Staubli VAL3: xyPut.pgx

program xyPut(num x_nX (dimensions=1), num x_nY (dimensions=1), string x_sKey (dimensions=1))
begin
  gotoxy(x_nX,x_nY)
  put(x_sKey)
end
